VAR_GLOBAL RETAIN
	productPoolSize : UDINT := 20;
	productKey : STRING := ' ';
END_VAR

(* stored: Version 1.1.0.1
   GVL G: Id {g} *)
